# EPICS autosave request: ttiEX355P/ttiEX355P_settings.req
$(P):CURRENT
$(P):OUTPUT
$(P):VOLTAGE
